RoboDK station: Programma schuine kant.rdk

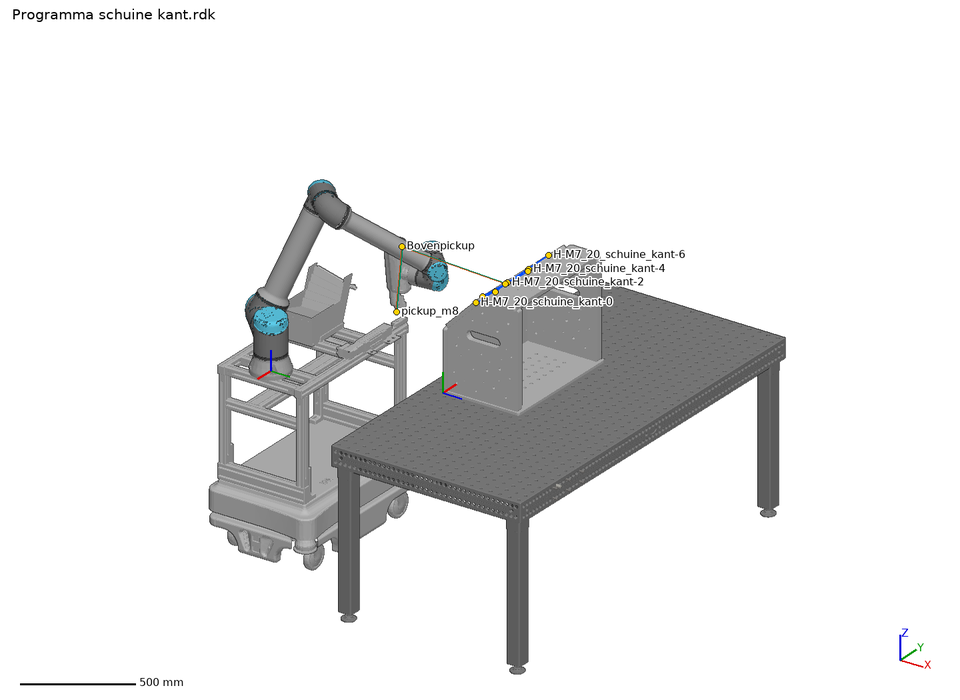
[picture v0: the station drawn from its stored meshes, robots at their saved joint values, targets as dots, program paths as lines]
Station Programma schuine kant (saved by RoboDK 5.7.0). Poses are relative to the parent item; angles as X-Y-Z fixed-axis rotations.
Station parameters (name, value as stored): CollisionFreePlanner, UR10e, CollisionFreePlanner-Rob UR10e
  - object Lastafel at (0, 0, 0) mm, size 1021.8 x 2000 x 842 mm
  - frame UR10e Base at (-1574.73, 215.14, 116.62) mm, rotated rx 0 ry 0 rz -90 deg
    - robot UR10e: 6 axes, payload 10 kg, reach 1300 mm, repeatability 0.05 mm, weight 28.9 kg
        modified DH rows (alpha deg, a mm, theta deg, d mm): 0, 0, 0, 180.7; 90, 0, 180, 0; 0, 612.6, 0, 0; 0, 571.335, 0, 174.15; -90, 0, 0, 119.85; 90, 0, 180, 116.55
        joint limits [-300, -150, -30, -360, -360, -360] to [300, 0, 180, 360, 360, 360]; home [30.872, -95.296, 116.362, -22.187, 121.11, 179.827]; saved at [-45.747, -65.18, 99.078, -38.37, -45.221, -90.148]
      - tool schroevendraaier all in met nieuw kopstuk en tool, TCP at (210, -1, 100.6) mm, rotated rx 90 ry -90 rz 90 deg, size 86.2 x 139.7 x 345.9 mm, geometry from schroevendraaier all in met nieuw kopstuk en tool.STEP
    - object Assembly mir + frame aangepast naar ur10e versie 2 at (-733.08, 277.19, -552.66) mm, rotated rx 90 ry 0 rz 0.45 deg, size 901.1 x 1139.6 x 580.4 mm, geometry from Assembly mir + frame aangepast naar ur10e versie 2.STEP
  - frame CSV Frame at (-919, 576, 49.99) mm, rotated rx 90 ry 0 rz 90.11 deg
    - object Test object at (0, 0.01, 0) mm, size 650 x 517 x 400 mm, geometry from Test object.STEP
    - target H-M7_20_schuine_kant-0 (Cartesian target) at (128.87, 405.62, 85.34) mm, rotated rx 0.81 ry -44.99 rz 88.86 deg; joints [-147.406, -79.902, 120.532, 269.875, -248.421, -114.1] of UR10e
    - target H-M7_20_schuine_kant-1 (Cartesian target) at (77.12, 476.89, 156.6) mm, rotated rx -2.65 ry -44.94 rz 93.75 deg; joints [-153.522, -82.266, 114.393, 278.792, -249.196, -109.628] of UR10e
    - target H-M7_20_schuine_kant-2 (Cartesian target) at (325.68, 432.59, 112.3) mm, rotated rx 40.89 ry 20.7 rz -22.21 deg; joints [-146.143, -50.783, 72.966, 157.815, -213.745, -224.999] of UR10e
    - target H-M7_20_schuine_kant-3 (Cartesian target) at (340.66, 360.36, 40.07) mm, rotated rx 40.89 ry -20.7 rz 22.21 deg; joints [-156.137, -50.658, 56.216, 80.363, -339.241, -216.533] of UR10e
    - target H-M7_20_schuine_kant-4 (Cartesian target) at (502.06, 421.99, 101.71) mm, rotated rx 40.89 ry 20.7 rz -22.21 deg; joints [-146.93, -76.828, 108.915, -56.814, -302.297, -117.069] of UR10e
    - target H-M7_20_schuine_kant-5 (Cartesian target) at (570.16, 369.5, 49.22) mm, rotated rx 42.87 ry 15.25 rz -15.83 deg; joints [-140.564, -45.12, 45.923, 33.563, -332.222, -164.044] of UR10e
    - target H-M7_20_schuine_kant-6 (Cartesian target) at (588.54, 468.7, 148.42) mm, rotated rx 43.86 ry 11.27 rz -11.49 deg; joints [-143.114, -48.956, 65.119, -171.159, -27.528, 23.668] of UR10e
    - target Face_Target_0 (Cartesian target) at (332.83, 418.62, 98.34) mm, rotated rx 34.79 ry 30.57 rz -36.21 deg; joints [-154.019, -70.39, 81.746, -84.456, -32.111, -54.521] of UR10e
    - target pickup_m8 (Cartesian target) at (296.95, 143.94, -451.18) mm, rotated rx 9.58 ry 86.75 rz -77.13 deg; joints [-45.747, -65.18, 99.078, -38.37, -45.221, -90.148] of UR10e
    - target Bovenpickup (Cartesian target) at (307.87, 458.95, -429.97) mm, rotated rx -139.66 ry 89.26 rz 129.81 deg; joints [-136.006, -63.802, 89.759, 154.828, 46.597, 89.992] of UR10e
  - Python program csv_importernewest (listed below)
  - Python program generatefaceapproaches (listed below)
  - Python program TargetFixer (listed below)
  - Python program Make_approaches_paths (listed below)
  - program Program_Face_0 (51 instructions, listed below)
  - program Program_Main (3 instructions, listed below)
  - program pickupToFaceTarget0 (5 instructions, listed below)
  - program FaceTarget0Topickup (7 instructions, listed below)
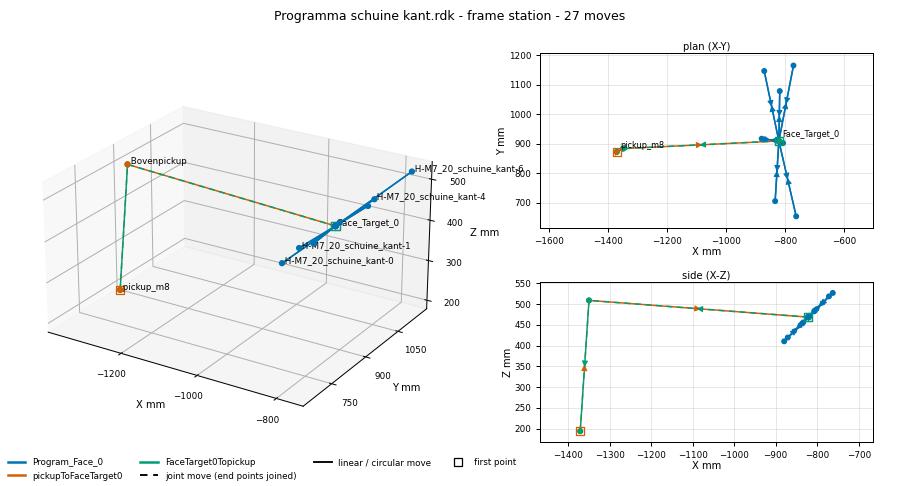
[picture p0: tool path of Programma schuine kant.rdk in frame station, 27 of 27 moves have a stored position in this frame; points joined in program order, loops and branches not executed]

--- Python program csv_importernewest ---
# This macro can load CSV files from Denso programs in RoboDK.
# Supported types of files are:
#  1-Tool data : Tool.csv
#  2-Work object data: Work.csv
#  3-Target data: P_Var.csv
# This macro can also filter a given targets file

# Type help("robodk.robolink") or help("robodk.robomath") for more information
# Press F5 to run the script
# Visit: http://www.robodk.com/doc/PythonAPI/
# For RoboDK API documentation

import os
import datetime

import tkinter as tk
from tkinter import messagebox

from robodk.robolink import *  # API to communicate with RoboDK
from robodk.robomath import *  # Robot toolbox
from robodk.robodialogs import *
from robodk.robofileio import *
import robodk.robolinkutils as RDKutils

DEBUG = False

debuglist = []

# Start communication with RoboDK
RDK = Robolink()

# Ask the user to select the robot
ROBOT = RDK.ItemUserPick('Select a robot', ITEM_TYPE_ROBOT)

# Check if the user selected a robot
if not ROBOT.Valid():
    quit()


# Ask the user to select a reference frame and get the active tool
BASE = ROBOT.Parent()
#BASE = RDK.Item('UR10e Base', ITEM_TYPE_FRAME)
#BASE = RDK.ItemUserPick('Select robot base frame', ITEM_TYPE_FRAME)
FRAME = RDK.ItemUserPick('Reference Frame', ITEM_TYPE_FRAME)
FRAMEPOSE = RDKutils.getPoseWrt(FRAME, BASE) #frame pose wrt robot base
TOOL = ROBOT.getLink(ITEM_TYPE_TOOL)
TOOLPOSE = RDKutils.getPoseWrt(TOOL, TOOL.Parent()) #tool pose wrt robot flange

if not FRAME.Valid() or not TOOL.Valid():
    raise Exception("Select appropriate FRAME and TOOL references")


# Function to convert XYZWPR to a pose
# Important! Specify the order of rotation
def xyzwpr_to_pose(xyzwpr):
    x, y, z, rx, ry, rz = xyzwpr
    return point_Zaxis_2_pose([x, y, z], [-rx, -ry, -rz])
    #return transl(x, y, z) * rotz(rz * pi / 180) * roty(ry * pi / 180) * rotx(rx * pi / 180)
    #return transl(x,y,z)*rotx(rx*pi/180)*roty(ry*pi/180)*rotz(rz*pi/180)
    #return KUKA_2_Pose(xyzwpr)


# csv_file = 'C:/Users/Albert/Desktop/Var_P.csv'
csv_file = getOpenFileName(RDK.getParam('PATH_OPENSTATION'))

# Specify file codec
codec = 'utf-8'  #'ISO-8859-1'


# Load P_Var.CSV data as a list of poses, including links to reference and tool frames
def load_targets(strfile):
    csvdata = LoadList(strfile, ',', codec)
    poses = []
    idxs = []
    for i in range(0, len(csvdata)):
        x, y, z, rx, ry, rz = csvdata[i][0:6]
        poses.append(xyzwpr_to_pose([x, y, z, rx, ry, rz]))
        #idxs.append(csvdata[i][6])
        idxs.append(i)

    return poses, idxs


# Load and display Targets from P_Var.CSV in RoboDK
def make_targets(strfile):
    poses, idxs = load_targets(strfile)
    program_name = getFileName(strfile)
    program_name = program_name.replace('-', '_').replace(' ', '_')

    for pose, idx in zip(poses, idxs):
        name = 'H-%s-%i' % (program_name, idx)
        target = RDK.Item(name, ITEM_TYPE_TARGET)
        if target.Valid():
            target.Delete()
        target = RDK.AddTarget(name, FRAME, ROBOT)


        target.setPose(pose)
        collision_free(target, idx)

def test_all_configurations(configurations):
    for joints in configurations:

        # turn collision checking off
        RDK.setCollisionActive(COLLISION_OFF)

        # move to target
        try:
            ROBOT.MoveJ(joints)
        except TargetReachError:
            continue

        # turn collision checking on, test for collisions
        RDK.setCollisionActive(COLLISION_ON)

        collision = RDK.Collisions()
        print(f"collision: {collision}")
        debuglist.append(f"collision: {collision}")

        collision_items = RDK.CollisionItems()
        if TOOL in collision_items or collision == 0:
            break

    try:
        collision
    except NameError:
        collision = -2
        print("Target cannot be reached or is to close to a singularity")
        debuglist.append("Target cannot be reached or is to close to a singularity")

    return collision


def test_collision_target(target, rz):
    if DEBUG:
        print("testing at target")
        debuglist.append("testing at target")

    possible_robot_configurations = ROBOT.SolveIK_All(target.Pose(), tool=TOOLPOSE, reference=FRAMEPOSE)
    issues_value = test_all_configurations(possible_robot_configurations) # returns 0 if at least one configuration is without issues

    return issues_value

def test_issues_point(target, rz, flip_approach=False):
    if DEBUG:
        print("testing point")
        debuglist.append("testing point")

    # Get the original pose
    original_pose = target.Pose()

    # For vertical walls, we might need to completely flip the approach
    if flip_approach:
        # Rotate 180 degrees around Y axis (assuming Y is the axis parallel to the wall)
        # This effectively approaches from the opposite direction
        target_new_pose = RelTool(original_pose, 0, 0, 0, 0, 180, 0)
        # Then apply the requested Z rotation
        target_new_pose = RelTool(target_new_pose, 0, 0, 0, 0, 0, rz)
    else:
        # Standard rotation around Z axis only
        target_new_pose = RelTool(original_pose, 0, 0, 0, 0, 0, rz)

    possible_robot_configurations = ROBOT.SolveIK_All(target_new_pose, tool=TOOLPOSE, reference=FRAMEPOSE)
    issues_value = test_all_configurations(possible_robot_configurations)

    return issues_value, target_new_pose

rotation_direction = "pos"
direction_changes = 0
holes_no_solution = []

def collision_free(target, idx):
    rotation_step = 30
    repmax = 360/rotation_step
    global rotation_direction
    global direction_changes
    s = 0
    rep = 0

    print(f"\nHole {idx}")
    debuglist.append(f"\nHole {idx}")

    # First try the original approach
    issues_value, target_new_pose = test_issues_point(target, 0, flip_approach=False)

    # If there's a collision, try different approaches
    while issues_value != 0 and s < 100:
        print(f"s before: {s}")
        debuglist.append(f"s before: {s}")
        print(f"rep: {rep}")
        debuglist.append(f"rep: {rep}")
        print(f"rotation direction: {rotation_direction}")
        debuglist.append(f"rotation direction: {rotation_direction}")
        print(f"direction changes: {direction_changes}")
        debuglist.append(f"direction changes: {direction_changes}")

        s += 1

        # For unreachable targets or potential vertical wall collision situations
        if issues_value == -2 and direction_changes < 2:
            if rotation_direction == "pos":
                rotation_direction = "neg"
                direction_changes += 1
                r = -1
            else:
                rotation_direction = "pos"
                direction_changes += 1
                r = 1

            # Try the opposite approach direction if we've changed direction once already
            # This is key for vertical walls
            if direction_changes >= 1:
                issues_value, target_new_pose = test_issues_point(target, r*rotation_step, flip_approach=True)
            else:
                issues_value, target_new_pose = test_issues_point(target, r*rotation_step, flip_approach=False)

            target.setPose(target_new_pose)

        # For collision situations, rotate around Z
        elif issues_value > 0 and rep < repmax:
            RDK.setCollisionActive(COLLISION_OFF) # collision off

            ROBOT.MoveJ(target.Pose())

            if rotation_direction == "neg":
                r = -1
            elif rotation_direction == "pos":
                r = 1

            # After trying several rotations, try the flip approach
            if rep > repmax/2:
                issues_value, target_new_pose = test_issues_point(target, r*rotation_step, flip_approach=True)
            else:
                issues_value, target_new_pose = test_issues_point(target, r*rotation_step, flip_approach=False)

            target.setPose(target_new_pose)
            rep += 1

        elif direction_changes >= 2 or rep >= repmax:
            break

        else:
            RDK.ShowMessage(f"Unknown error occured at Hole {idx} while looking for collision free position")

    direction_changes = 0
    if issues_value == 0:
        print(f"No issues at Hole {idx}")
        debuglist.append(f"No issues at Hole {idx}")
    elif direction_changes >= 2 or rep >= repmax or s >= 100:
        RDK.ShowMessage(f"No solution found for Hole {idx}", False)
        holes_no_solution.append(idx)

        print(f"No solution found for Hole {idx}")
        debuglist.append(f"No solution found for Hole {idx}")

    else:
        RDK.ShowMessage(f"Unknown error occured at Hole {idx} while looking for collision free position")

        print(f"Unknown error occured at Hole {idx} while looking for collision free position")
        debuglist.append(f"Unknown error occured at Hole {idx} while looking for collision free position")


MAKE_GUI_PROGRAM = True

ROBOT.setFrame(FRAME)
ROBOT.setTool(TOOL)

if RDK.RunMode() == RUNMODE_SIMULATE:
    MAKE_GUI_PROGRAM = True
    # MAKE_GUI_PROGRAM = mbox('Do you want to create a new program? If not, the robot will just move along the targets', 'Yes', 'No')
else:
    # if we run in program generation mode just move the robot
    MAKE_GUI_PROGRAM = False

if MAKE_GUI_PROGRAM:
    RDK.Render(False)  # Faster if we turn render off
    make_targets(csv_file)
else:
    l

if len(holes_no_solution) != 0:
    RDK.ShowMessage(f"Holes without solution: {holes_no_solution}")

if DEBUG:
    print(f"Holes without solution: {holes_no_solution}")
    debuglist.append(f"Holes without solution: {holes_no_solution}")

    current_time = datetime.datetime.now()
    filename = os.path.splitext(os.path.basename(__file__))
    with open("C:/Users/Laura/Documents/1.Windesheim/Stage/2024/Lectoraat/Deelvragen/2.Targets maken/debugfile.txt", "a") as file:
        file.write("\n\n-----------------------------------------------\n")
        file.write(current_time.strftime("%c"))
        file.write("\n-----------------------------------------------\n")
        for prints in debuglist:
            file.write(prints)
            file.write("\n")
        file.write(holes_no_solution)
        file.write(filename[0])

--- Python program generatefaceapproaches ---
from robodk.robolink import *  # API to communicate with RoboDK
from robodk.robomath import *   # Robot toolbox
import robodk.robolinkutils as RDKutils
from robodk import robolink

DEBUG = False

# Link to RoboDK
RDK = Robolink()

ROBOT = RDK.ItemUserPick('Select a Robot', ITEM_TYPE_ROBOT)
FRAME = RDK.ItemUserPick('Reference Frame', ITEM_TYPE_FRAME)

if not ROBOT.Valid() or not FRAME.Valid():
    raise Exception("Select appropriate ROBOT and FRAME")

BASE = RDK.Item('UR10e Base', ITEM_TYPE_FRAME)
FRAMEPOSE = RDKutils.getPoseWrt(FRAME, BASE)  # frame pose with respect to robot base
TOOL = ROBOT.getLink(ITEM_TYPE_TOOL)
TOOLPOSE = RDKutils.getPoseWrt(TOOL, TOOL.Parent())  # tool pose with respect to robot flange

# Get all the holes as targets (only those with "H" in the name)
All_items = RDK.ItemList(ITEM_TYPE_TARGET)
RDK_items = [item for item in All_items if "H" in item.Name()]
print(f"Holes: {len(RDK_items)}")

RDK.setCollisionActive(COLLISION_OFF)

def print_xyzrpw(pose):
    x, y, z, rx, ry, rz = pose_2_xyzrpw(pose)
    print(x, y, z, rx, ry, rz)

class Hole:
    def __init__(self, pose, target):
        self.pose = pose
        self.target = target
        self.name = self.target.Name()
        self.split_position_rotation(pose)

    def split_position_rotation(self, pose):
        x, y, z, rx, ry, rz = pose_2_xyzrpw(pose)
        self.position = (x, y, z)
        # Get the z-axis direction (3rd column of the rotation matrix)
        self.rotation = pose[0:3, 2]
        zfacing1 = round(self.rotation.tolist()[0])
        zfacing2 = round(self.rotation.tolist()[1])
        zfacing3 = round(self.rotation.tolist()[2])
        self.rot_identifier = f"{zfacing1}_{zfacing2}_{zfacing3}"

class Face:
    def __init__(self, key):
        self.key = key
        self.get_midpoint(key)
        self.rotation = self.holes[0].rotation.tolist()
        self.offset_multiplier = self.rotation
        self.approaches = []  # Not used in the new functions

    def get_midpoint(self, key):
        # Retrieve all holes corresponding to this face
        self.holes = dic[key]
        x_values = [hole.position[0] for hole in self.holes]
        y_values = [hole.position[1] for hole in self.holes]
        z_values = [hole.position[2] for hole in self.holes]

        # Sort and compute the midpoint as the average of the min and max values
        x_values.sort()
        y_values.sort()
        z_values.sort()
        min_x, max_x = x_values[0], x_values[-1]
        min_y, max_y = y_values[0], y_values[-1]
        min_z, max_z = z_values[0], z_values[-1]

        mid_x = (min_x + max_x) / 2
        mid_y = (min_y + max_y) / 2
        mid_z = (min_z + max_z) / 2

        self.midpoint = (mid_x, mid_y, mid_z)

        # Use the first hole's pose as a template and update its translation to the midpoint
        self.ref_hole = self.holes[0]
        ref_pose = self.ref_hole.pose
        ref_pose[0, 3] = mid_x
        ref_pose[1, 3] = mid_y
        ref_pose[2, 3] = mid_z
        self.midpose = ref_pose

    def add_approaches(self, approach):
        self.approaches.append(approach)

# --- Process holes and group them into faces based on z-axis orientation ---
holes = []
dic = {}
faces = []

# Convert the target items into Hole objects
for item in RDK_items:
    hole = Hole(item.Pose(), item)
    holes.append(hole)

# Group holes with the same z-axis orientation (rounded)
for hole in holes:
    if hole.rot_identifier in dic:
        dic[hole.rot_identifier].append(hole)
    else:
        dic[hole.rot_identifier] = [hole]

# Create Face objects from the groups
for key in dic:
    face = Face(key)
    faces.append(face)

# --- NEW FUNCTION: Create face targets at the midpoint of each face ---
def create_face_targets():
    """
    For each computed face, create a new target in RoboDK at the face midpoint.
    """
    for i, face in enumerate(faces):
        face_target_name = f"Face_Target_{i}"

        # Delete existing target if it exists
        existing_target = RDK.Item(face_target_name, ITEM_TYPE_TARGET)
        if existing_target.Valid():
            existing_target.Delete()

        # Start with the original midpose
        collision_free_pose = face.midpose.copy()
        collision_found = True

        print(f"Checking collision for face {i} at midpoint {face.midpoint}")

        # Enable collision detection
        RDK.setCollisionActive(COLLISION_ON)

        # First try the original pose (0 degrees)
        ROBOT.setPose(face.midpose)
        collision = RDK.Collisions()

        if collision == 0:
            collision_free_pose = face.midpose
            collision_found = False
            print(f"Found collision-free pose for face {i} with rz = 0 degrees")
        else:
            # Try alternating positive and negative rotations
            rotation_step = 10
            max_rotation = 720

            while collision_found and rotation_step <= max_rotation:
                # Try both positive and negative rotations for this step
                for rotation_direction in ["pos", "neg"]:
                    if rotation_direction == "neg":
                        r = -1
                    elif rotation_direction == "pos":
                        r = 1

                    rz = r * rotation_step
                    test_pose = RelTool(face.midpose, 0, 0, 0, 0, 0, rz)

                    # Set robot to test pose and check for collision
                    ROBOT.setPose(test_pose)
                    collision = RDK.Collisions()

                    if collision == 0:
                        # No collision found - we can use this pose
                        collision_free_pose = test_pose
                        collision_found = False
                        print(f"Found collision-free pose for face {i} with rz = {rz} degrees")
                        break
                    else:
                        print(f"Collision detected for face {i} at rz = {rz}, continuing search...")

                # If collision-free pose found, break out of the while loop
                if not collision_found:
                    break

                # Increment rotation step for next iteration
                rotation_step += 10

        if collision_found:
            print(f"Warning: Could not find collision-free pose for face {i} after full rotation (±{max_rotation}°)")
            # Use original pose anyway
            collision_free_pose = face.midpose

        # Create the face target with the collision-free pose
        face_target = RDK.AddTarget(face_target_name, FRAME, ROBOT)
        face_target.setPose(collision_free_pose)

        print(f"Created face target for face {i} at midpoint {face.midpoint}")

    # Turn off collision detection when done
    RDK.setCollisionActive(COLLISION_OFF)



# --- NEW FUNCTION: Create a program for each face using MoveL commands ---
def create_face_programs():
    """
    For each face, generate a program that moves from the face target (approach target)
    to every hole target on that face using a MoveL command.
    Each move from the face target to a hole target is followed by a return move to the face target.
    """

    for i, face in enumerate(faces):
        face_target_name = f"Face_Target_{i}"
        face_target = RDK.Item(face_target_name, ITEM_TYPE_TARGET)
        prog_name = f"Program_Face_{i}"
        existing_prog = RDK.Item(prog_name, ITEM_TYPE_PROGRAM)
        if existing_prog.Valid():
            existing_prog.Delete()
        prog = RDK.AddProgram(prog_name, ROBOT)

        # Add a move to the face target as the starting (approach) move


        # For each hole in this face, add a MoveL to go to the hole target and then a MoveL back to the face target.
        for j, hole in enumerate(face.holes):  # Use enumerate to get the index 'j' of the hole

            # Construct the program names using f-strings
            program_to_call_2 = f'pickupToFaceTarget{i}'
            program_to_call_1 = f'FaceTarget{i}Topickup'

            if j == 0:
                prog.RunInstruction(program_to_call_2, robolink.INSTRUCTION_CALL_PROGRAM)

            prog.MoveL(face_target)
            prog.MoveL(hole.target)

            prog.RunInstruction('screw_in(20)', robolink.INSTRUCTION_CALL_PROGRAM)  # Tighten screw
            prog.RunInstruction('screw_out(0)', robolink.INSTRUCTION_CALL_PROGRAM)  # Release screwdriver

            prog.MoveL(face_target)

            prog.RunInstruction(program_to_call_1, robolink.INSTRUCTION_CALL_PROGRAM)

            # Check if it's NOT the last hole in the face
            if j < len(face.holes) - 1:

                prog.RunInstruction(program_to_call_2, robolink.INSTRUCTION_CALL_PROGRAM)

            print(f"Program {prog_name}: Added MoveL from approach target to hole {hole.name} and back.")

def addmainprogram():


    prog_name = f"Program_Main"
    existing_prog = RDK.Item(prog_name, ITEM_TYPE_PROGRAM)
    if existing_prog.Valid():
        existing_prog.Delete()
    prog = RDK.AddProgram(prog_name, ROBOT)


    # set reference frame
    # set tcp
    prog.setTool(RDK.ItemUserPick('Select tool', ITEM_TYPE_TOOL))
    prog.setFrame(RDK.ItemUserPick('Select frame', ITEM_TYPE_FRAME))

    # Voeg elke program toe aan een groot programma die met "program_face" begint
    for j in range(len(faces)):
        sub_prog_name = f"Program_Face_{j}"
        prog.RunInstruction(sub_prog_name)



def generate_pickup_links():

    # for i, face in enumerate(faces):
    #     ROBOT.setPoseFrame(face.midpose[i]) ## deze lijn
    #     status = RDK.PluginCommand("CollisionFreePlanner", "Add")
    #     print(status)

    # Define the name that is given in RoboDK for the pickup target
    pickup_target_name = "pickup"  # The name of the target in your RoboDK station

    # Get the actual RoboDK Item for the pickup target
    Target_Pickup_item = RDK.Item(pickup_target_name, ITEM_TYPE_TARGET)

    if not Target_Pickup_item.Valid():
        print(
            f"Error: Pickup target '{pickup_target_name}' not found in RoboDK station. Skipping pickup link generation.")
        return  # Exit the function if the pickup target doesn't exist

    # For every face, create 2 planned motions (programs)
    # One from Face_Target_i to 'pickup' target
    # One from 'pickup' target to Face_Target_i
    for i, face in enumerate(faces):  # Iterate through faces to get the numerical index 'i'
        # Get the name of the Face_Target for the current face
        face_target_name = f"Face_Target_{i}"

        # Define the names for the programs to be created by the plugin
        program_name_to_pickup = f"FaceTarget{i}Topickup"
        program_name_from_pickup = f"pickupToFaceTarget{i}" # Corrected: consistency with previous example

        # --- Check and delete existing "To Pickup" program ---
        existing_prog_to_pickup = RDK.Item(program_name_to_pickup, ITEM_TYPE_PROGRAM)
        if existing_prog_to_pickup.Valid():
            print(f"Deleting existing program: {program_name_to_pickup}")
            existing_prog_to_pickup.Delete()

        print(f"Attempting to join: {face_target_name} to {pickup_target_name} as {program_name_to_pickup}")

        # Call the plugin command to join the face target to the pickup target
        status_to_pickup = RDK.PluginCommand(
            "CollisionFreePlanner",
            "Join",
            f"{face_target_name}|{pickup_target_name}|{program_name_to_pickup}"
            )
        print(f"Status for '{program_name_to_pickup}': {status_to_pickup}")

        # --- Check and delete existing "From Pickup" program ---
        existing_prog_from_pickup = RDK.Item(program_name_from_pickup, ITEM_TYPE_PROGRAM)
        if existing_prog_from_pickup.Valid():
            print(f"Deleting existing program: {program_name_from_pickup}")
            existing_prog_from_pickup.Delete()

        print(f"Attempting to join: {pickup_target_name} to {face_target_name} as {program_name_from_pickup}")

        # Call the plugin command to join the pickup target to the face target
        status_from_pickup = RDK.PluginCommand(
            "CollisionFreePlanner",
            "Join",
            f"{pickup_target_name}|{face_target_name}|{program_name_from_pickup}"
             )
        print(f"Status for '{program_name_from_pickup}': {status_from_pickup}")


    print("\nPickup link generation process finished.")

#def generate_unscrewing_programs():


# --- Main execution: Run only the new functions ---
if __name__ == '__main__':
    create_face_targets()
    generate_pickup_links()
    create_face_programs()
    addmainprogram()

#for documentation of the collision free motion planner see https://robodk.com/addin/com.robodk.plugin.collisionfreeplanner, searched ages for API documentation

--- Python program TargetFixer ---
from robodk import robolink, robomath
import robodk.robolinkutils as RDKutils

from robodk.robolink import *       # RoboDK API
from robodk.robomath import *        # Math toolbox (provides transl, etc.)
from robodk.robodialogs import *
from robodk.robofileio import *

def main():
    # Initialize RoboDK instance
    RDK = robolink.Robolink()

    # Let the user pick a Robot and a Reference Frame
    ROBOT = RDK.ItemUserPick('Select a Robot', ITEM_TYPE_ROBOT)
    FRAME = RDK.ItemUserPick('Select a Reference Frame', ITEM_TYPE_FRAME)
    if not ROBOT.Valid() or not FRAME.Valid():
        raise Exception("Select appropriate ROBOT and FRAME")

    # Get Base, Tool and FRAME pose (adjust names as needed)
    BASE = RDK.Item('UR10e Base', ITEM_TYPE_FRAME)
    FRAMEPOSE = RDKutils.getPoseWrt(FRAME, BASE) if BASE.Valid() else FRAME.Pose()
    TOOL = ROBOT.getLink(ITEM_TYPE_TOOL)
    TOOLPOSE = RDKutils.getPoseWrt(TOOL, TOOL.Parent())

    # Activate collision checking
    RDK.setCollisionActive(COLLISION_ON)

    # Get all targets (or filter them as needed)
    all_targets = RDK.ItemList(ITEM_TYPE_TARGET)

    fixed_targets = []
    unfixed_targets = []

    # Process every target one by one
    for target in all_targets:
        original_pose = target.Pose()
        print(f"\nProcessing target: {target.Name()}")

        # First, check if the target is already collision free:
        if not target_in_collision(RDK, ROBOT, target, FRAMEPOSE, TOOLPOSE):
            print(f"Target {target.Name()} is already collision free. No fix needed.")
            continue

        print(f"Target {target.Name()} is in collision. Attempting to fix by shifting along principal axes...")

        # Try to fix by shifting along X, then Y, then Z
        fixed = fix_target(target, original_pose, RDK, ROBOT, FRAMEPOSE, TOOLPOSE)
        if fixed:
            fixed_targets.append(target.Name())
        else:
            unfixed_targets.append(target.Name())
            target.setPose(original_pose)  # revert to original if no fix was found

    # Summary report
    print("\nTarget fixing complete.")
    print("Fixed targets:")
    for t in fixed_targets:
        print("  -", t)
    if unfixed_targets:
        print("Targets that could not be fixed:")
        for t in unfixed_targets:
            print("  -", t)

def target_in_collision(RDK, ROBOT, target, FRAMEPOSE, TOOLPOSE):
    """
    Checks whether the given target causes a collision.
    It does so by attempting to solve IK and simulating a MoveJ.
    Returns True if a collision (or no valid configuration) is detected.
    """
    pose = target.Pose()
    possible_configs = ROBOT.SolveIK_All(pose, tool=TOOLPOSE, reference=FRAMEPOSE)
    if not possible_configs:
        return True
    for joints in possible_configs:
        try:
            ROBOT.MoveJ(joints)
        except Exception:
            continue
        if not RDK.Collisions():
            return False
    return True

def fix_target(target, original_pose, RDK, ROBOT, FRAMEPOSE, TOOLPOSE):
    """
    Attempts to fix a target by shifting it along each principal axis.

    For each axis (X, Y, Z), the function:
      - Tries a positive shift in 10-mm increments (10 steps).
      - Reverts to the original pose.
      - Tries a negative shift in 10-mm increments (10 steps).

    If a collision-free pose is found during any of these tests, the target is updated.
    Returns True if a valid pose is found, otherwise False.
    """
    # Define axes along which to shift using lambda functions that generate translation matrices.
    # The transl(x, y, z) function creates a translation matrix in the local coordinate system when multiplied with a pose.
    axes = [
        ("X", lambda d: transl(d, 0, 0)),
        ("Y", lambda d: transl(0, d, 0)),
        ("Z", lambda d: transl(0, 0, d))
    ]

    # For each axis...
    for axis_name, shift_func in axes:
        # Try positive direction shifts first
        for i in range(1, 11):
            shift_matrix = shift_func(10 * i)  # 10-mm increments
            test_pose = original_pose * shift_matrix
            target.setPose(test_pose)
            if not target_in_collision(RDK, ROBOT, target, FRAMEPOSE, TOOLPOSE):
                print(f"Target {target.Name()} fixed with a +{10*i} mm shift along {axis_name}.")
                return True
        # Revert to the original pose before trying the negative direction
        target.setPose(original_pose)
        for i in range(1, 11):
            shift_matrix = shift_func(-10 * i)
            test_pose = original_pose * shift_matrix
            target.setPose(test_pose)
            if not target_in_collision(RDK, ROBOT, target, FRAMEPOSE, TOOLPOSE):
                print(f"Target {target.Name()} fixed with a {-10*i} mm shift along {axis_name}.")
                return True
        # Revert to the original pose before trying the next axis
        target.setPose(original_pose)
    return False

if __name__ == '__main__':
    main()

--- Python program Make_approaches_paths ---
from robodk.robolink import *  # API to communicate with RoboDK
from robodk.robomath import *  # Robot toolbox
import robodk.robolinkutils as RDKutils


DEBUG = False


# Link to RoboDK
RDK = Robolink()

ROBOT = RDK.ItemUserPick('Select a Robot', ITEM_TYPE_ROBOT)
FRAME = RDK.ItemUserPick('Reference Frame', ITEM_TYPE_FRAME)

if not ROBOT.Valid() or not FRAME.Valid():
    raise Exception("Select appropriate ROBOT and FRAME")

BASE = RDK.Item('UR10e Base', ITEM_TYPE_FRAME)
#BASE = RDK.ItemUserPick('Select robot base frame', ITEM_TYPE_FRAME)
FRAMEPOSE = RDKutils.getPoseWrt(FRAME, BASE) #frame pose wrt robot base
TOOL = ROBOT.getLink(ITEM_TYPE_TOOL)
TOOLPOSE = RDKutils.getPoseWrt(TOOL, TOOL.Parent()) #tool pose wrt robot flange




# get all the holes as items
All_items = RDK.ItemList(ITEM_TYPE_TARGET)
#RDK_items = [item for item in All_items if "Hole" in item.Name()]
RDK_items = [item for item in All_items if "H" in item.Name()]
print(f"Holes: {len(RDK_items)}")

RDK.setCollisionActive(COLLISION_OFF)

def print_xyzrpw(pose):
    x, y, z, rx, ry, rz = pose_2_xyzrpw(pose)
    print(x, y, z, rx, ry, rz)


class Hole:
    def __init__(self, pose, target):
        self.pose = pose
        self.target = target
        self.name = self.target.Name()
        self.split_position_rotation(pose)

    def split_position_rotation(self, pose):
        x, y, z, rx, ry, rz = pose_2_xyzrpw(pose)
        self.position = x, y, z
        # get the way the z-axis is facing
        self.rotation = pose[0:3,2] # from all 3 rows (0:3) only the 3rd column (index 2) (the last column of the rotation matrix)
        # format the z-axis facing, so it can be made a key in the dictonary
        zfacing1 = round(self.rotation.tolist()[0])
        zfacing2 = round(self.rotation.tolist()[1])
        zfacing3 = round(self.rotation.tolist()[2])
        self.rot_identifier = f"{zfacing1}_{zfacing2}_{zfacing3}"

class Face:
    def __init__(self, key):
        self.key = key
        self.get_midpoint(key)
        self.rotation = self.holes[0].rotation.tolist()
        self.offset_multiplier = self.rotation
        self.approaches = []

    def get_midpoint(self, key):
        #global dic
        #targets from key
        self.holes = dic[key]
        #x, y, z from targets
        self.x_values = []
        self.y_values = []
        self.z_values = []
        for hole in self.holes:
            x, y, z = hole.position
            self.x_values.append(x)
            self.y_values.append(y)
            self.z_values.append(z)
        if DEBUG:
            print("ranges:")
            print(self.x_values)
            print(self.y_values)
            print(self.z_values)
        #min and max of these
        self.x_values.sort()
        min_x = self.x_values[0]
        max_x = self.x_values[len(self.x_values)-1]
        offset_x = (max_x - min_x)/2
        mid_x = max_x - offset_x
        self.xranges = min_x, max_x, mid_x

        self.y_values.sort()
        min_y = self.y_values[0]
        max_y = self.y_values[len(self.y_values)-1]
        offset_y = (max_y - min_y)/2
        mid_y = max_y - offset_y
        self.yranges = min_y, max_y, mid_y

        self.z_values.sort()
        min_z = self.z_values[0]
        max_z = self.z_values[len(self.z_values)-1]
        offset_z = (max_z - min_z)/2
        mid_z = max_z - offset_z
        self.zranges = min_z, max_z, mid_z

        self.midpoint = mid_x, mid_y, mid_z

        self.ref_hole = self.holes[0]
        ref_pose = self.ref_hole.pose
        ref_pose[0,3] = mid_x
        ref_pose[1,3] = mid_y
        ref_pose[2,3] = mid_z
        self.midpose = ref_pose
        if DEBUG:
            print("min, max, mid: ")
            print("x: ", self.xranges)
            print("y: ", self.yranges)
            print("z: ", self.zranges)
            print("midpoint: ", self.midpoint)
            print("midpose: ", self.midpose)

    def add_approaches(self, approach):
        self.approaches.append(approach)



class Approach:
    def __init__(self, face, number):
        self.face = face
        self.number = number
        self.target = self.make_approach_target(face, number)

    def make_approach_target(self, face, number):
        approach_point = self.get_approach_point(face)
        approach_target = RDK.Item(f"approach {idx} {face.rotation}", ITEM_TYPE_TARGET)
        if approach_target.Valid():
            approach_target.Delete()
        approach_target = RDK.AddTarget(f"approach {idx} {face.rotation}", FRAME, ROBOT)
        approach_target.setPose(approach_point)
        if DEBUG:
            print("approach target:\n", approach_point)
        return approach_target

    def get_approach_point(self, face):
        MAX_APPROACH = 100 #in mm
        MIN_APPROACH = 20 #in mm
        STEP = 40 #in mm
        ROT_STEP = 20 #in degrees
        approach_point = self.test_distance(face, MAX_APPROACH, MIN_APPROACH, STEP, ROT_STEP)
        return approach_point

    def test_distance(self, face, MAX_APPROACH, MIN_APPROACH, STEP, ROT_STEP):
        approach_distance = MAX_APPROACH
        rep = 0
        repmax = 360/ROT_STEP
        rot_offset = 0
        rotation_direction = "pos"
        direction_changes = 0

        z = approach_distance
        issues, approach_point = self.test_point(face.midpose, z, 0)
        #first_issues_value = issues
        if issues == -2:
            rz = 180
            rot_offset = rz
            issues, approach_point = self.test_point(face.midpose, z, rz)

        sa = 0
        while issues != 0 and approach_distance >= MIN_APPROACH + STEP and sa < 100:
            sa += 1
            approach_distance -= STEP
            z = approach_distance
            rz = 0
            issues, approach_point = self.test_point(face.midpose, z, rz)
            issues, approach_point = self.rotate(face, issues, approach_distance, rot_offset, ROT_STEP)

        return approach_point

    def rotate(self, face, issues, approach_distance, rot_offset, ROT_STEP):
        repmax = 360/ROT_STEP
        rotation_direction = "pos"
        direction_changes = 0
        rep = 0
        sb = 0
        while issues != 0 and sb < 100:
            sb += 1
            if issues == -2 and direction_changes < 2:
                if rotation_direction == "pos":
                    rotation_direction = "neg"
                    r = -1 #rotation factor to make the rotation negative
                else:
                    rotation_direction = "pos"
                    r = 1
                direction_changes += 1
                z = approach_distance
                rz = rot_offset + r * ROT_STEP
                issues, approach_point = self.test_point(face.midpose, z, rz)
            elif issues > 0 and rep < repmax:
                if rotation_direction == "neg":
                    r = -1
                else:
                    r = 1
                rep += 1
                z = approach_distance
                rz = rot_offset + r * ROT_STEP
                rot_offset = rz
                issues, approach_point = self.test_point(face.midpose, z, rz)
            elif direction_changes >= 2 or rep >= repmax:
                break

            else:
                print(f"Unknown error occured at Approach {self.number}")

        if issues != 0 and (direction_changes >= 2 or rep >= repmax or sb == 100):
            print(f"No solution found for Approach {self.number}")
            global approach_noSolution
            approach_noSolution.append(self.number)
            RDK.ShowMessage(f"No solution found for Approach {self.number}", False)
        return issues, approach_point

    def test_point(self, point, z, rz):
        # define the position to test for collisions
        test_point = RelTool(point, 0,0,z, 0,0,rz)
        possible_robot_configurations = ROBOT.SolveIK_All(test_point, tool=TOOLPOSE, reference=FRAMEPOSE)
        issues = self.test_all_configurations(possible_robot_configurations)
        return issues, test_point

    def test_all_configurations(self, configurations):
        for joints in configurations:

            # turn collision checking off
            RDK.setCollisionActive(COLLISION_OFF)
            is_active = RDK.Command("CollisionActive")
            #print(f"collsion active? should be off (0) {is_active}")

            # move to target
            try:
                ROBOT.MoveJ(joints)
            except TargetReachError:
                continue

            # turn collision checking on, test for collisions
            RDK.setCollisionActive(COLLISION_ON)
            is_active = RDK.Command("CollisionActive")
            #print(f"collsion active? should be on (1) {is_active}")
            collision = RDK.Collisions()
            #print(f"collision: {collision}")
            collision_items = RDK.CollisionItems()
            if TOOL in collision_items or collision == 0:
                break

        try:
            collision
        except NameError:
            collision = -2 # TargetReachError occures for every configuration
            #print("Target cannot be reached or is to close to a singularity")

        return collision

def collision_free_paths(face, approach):
    possible_configurations = ROBOT.SolveIK_All(approach.target.Pose(), tool=TOOLPOSE, reference=FRAMEPOSE)
    for i, joints in enumerate(possible_configurations):
        print(f"testing configuration {i+1}")
        for j, hole in enumerate(face.holes):
            RDK.setCollisionActive(COLLISION_OFF)
            ROBOT.MoveJ(joints)
            RDK.setCollisionActive(COLLISION_ON)
            issues = ROBOT.MoveJ_Test(joints, hole.target.Joints())
            print(f"Hole {hole.name} with issues = {issues}")
            if issues == 0:
                continue
            break

        if issues == 0:
            print(f"found valid configuration: {i+1}")
            approach.target.setJoints(joints)
            break

    if issues != 0:
        print(f"no configuration found for approach {approach.number}")
        path_no_solution.append(hole.name)

holes = []
dic = {}
faces = []
approach_noSolution = []
path_no_solution = []

# convert the target items into target objects
for item in RDK_items:
    hole = Hole(item.Pose(), item)
    holes.append(hole)

# put the targets with the z-axis facing the same way together
for hole in holes:
    if hole.rot_identifier in dic:
        #dic exists put it in
        dic[hole.rot_identifier].append(hole)
    else:
        #make a dic and put it in
        dic[hole.rot_identifier] = [hole]

keys = list(dic.keys())
for key in keys:
    if DEBUG:
        print(f"{key}: {dic[key]}")
    face = Face(key)
    faces.append(face)
    if DEBUG:
        print(face.midpoint)

for idx, face in enumerate(faces):
    if DEBUG:
        print(faces)
    approach = Approach(face, idx)
    face.add_approaches(approach)

    #paden maken tussen approach en targets die daar bij horen
    for approach in face.approaches:
        collision_free_paths(face, approach)
        for hole in face.holes:
            program_name = f"to {hole.name}"
            program = RDK.Item(program_name, ITEM_TYPE_PROGRAM)
            if program.Valid():
                program.Delete()
            program = RDK.AddProgram(program_name, ROBOT)
            ROBOT.MoveJ(approach.target)
            program.MoveJ(hole.target)

--- program Program_Face_0 (robot UR10e) ---
  Call screw_in(30)
  Call screw_out(0)
  Call pickupToFaceTarget0
  MoveL (Face_Target_0)
  MoveL (H-M7_20_schuine_kant-0)
  Call screw_in(30)
  Call screw_out(0)
  MoveL (Face_Target_0)
  Call FaceTarget0Topickup
  Call pickupToFaceTarget0
  MoveL (Face_Target_0)
  MoveL (H-M7_20_schuine_kant-1)
  Call screw_in(30)
  Call screw_out(0)
  MoveL (Face_Target_0)
  Call FaceTarget0Topickup
  Call pickupToFaceTarget0
  MoveL (Face_Target_0)
  MoveL (H-M7_20_schuine_kant-2)
  Call screw_in(30)
  Call screw_out(0)
  MoveL (Face_Target_0)
  Call FaceTarget0Topickup
  Call pickupToFaceTarget0
  MoveL (Face_Target_0)
  MoveL (H-M7_20_schuine_kant-3)
  Call screw_in(30)
  Call screw_out(0)
  MoveL (Face_Target_0)
  Call FaceTarget0Topickup
  Call pickupToFaceTarget0
  MoveL (Face_Target_0)
  MoveL (H-M7_20_schuine_kant-4)
  Call screw_in(30)
  Call screw_out(0)
  MoveL (Face_Target_0)
  Call FaceTarget0Topickup
  Call pickupToFaceTarget0
  MoveL (Face_Target_0)
  MoveL (H-M7_20_schuine_kant-5)
  Call screw_in(30)
  Call screw_out(0)
  MoveL (Face_Target_0)
  Call FaceTarget0Topickup
  Call pickupToFaceTarget0
  MoveL (Face_Target_0)
  MoveL (H-M7_20_schuine_kant-6)
  Call screw_in(30)
  Call screw_out(0)
  MoveL (Face_Target_0)
  Call FaceTarget0Topickup

--- program Program_Main (robot UR10e) ---
  Set Tool: schroevendraaier all in met nieuw kopstuk en tool
  Set Ref.: CSV Frame
  Call Program_Face_0

--- program pickupToFaceTarget0 (robot UR10e) ---
  Set Ref.: CSV Frame
  Set Tool: schroevendraaier all in met nieuw kopstuk en tool
  MoveJ (pickup_m8)
  MoveJ (Bovenpickup)
  MoveL (Face_Target_0)

--- program FaceTarget0Topickup (robot UR10e) ---
  Set Ref.: CSV Frame
  Set Tool: schroevendraaier all in met nieuw kopstuk en tool
  MoveJ (Face_Target_0)
  MoveJ (Bovenpickup)
  MoveL (pickup_m8)
  Call screw_in(30)
  Call screw_out(0)
